% RSLogix 500 project LINCE050116_TOP.RSS, saved by version 11.00.00.00 %
PROJECT "LINCETOP"    % processor: MicroLogix 1400 %

PROGRAM FILES
  LAD 2 "MAIN"  12 rungs  % Main Program Routine %
  LAD 70 "OFFSETS"  43 rungs
  LAD 88 "TIMESWITCH"  2 rungs
  LAD 89 "SECONDS"  2 rungs
  LAD 90 "HSC"  9 rungs
  LAD 99 "HMI SET"  3 rungs
  LAD 100 "STI"  55 rungs
  LAD 102 "SPEED"  6 rungs
  LAD 104 "P ADJUST"  8 rungs
  LAD 110 "SHIFT"  11 rungs
  LAD 120 "XFER IN"  3 rungs
  LAD 121 "SIM PARTS"  7 rungs
  LAD 122 "PARTDETECT"  12 rungs
  LAD 123 "OPTICWIDTH"  7 rungs
  LAD 124 "PART GAP"  8 rungs
  LAD 125 "OPTIC CL"  4 rungs
  LAD 126 "ALIGNMENT"  6 rungs
  LAD 127 "OPTIC_LOAD"  3 rungs
  LAD 128 "FELL PART"  12 rungs
  LAD 130 "INS 5 TRIG"  14 rungs
  LAD 131 "INS 5 RSLT"  18 rungs
  LAD 140 "INS 6 TRIG"  9 rungs
  LAD 141 "INS 6 RSLT"  18 rungs
  LAD 150 "INS 7 TRIG"  9 rungs
  LAD 151 "INS 7 RSLT"  18 rungs
  LAD 170 "PASSBLOW"  12 rungs
  LAD 180 "RECERK"  10 rungs
  LAD 200 "PRODRATE"  1 rungs
  LAD 230 "HMI GET"  1 rungs

DATA FILES
  O0 OUTPUT  6 elements
  I1 INPUT  8 elements
  S2 STATUS  66 elements
  B3 BINARY  14 elements
  T4 TIMER  40 elements
  C5 COUNTER  1 elements
  R6 CONTROL  14 elements
  N7 INTEGER  200 elements
  F8 FLOAT  100 elements
  B9 TOP BS DAT  256 elements
  B10 TEMP  128 elements  % temp for program change %
  B11 TOP ER DAT  256 elements
  N12 TEMP  128 elements  % until sort out program io difference %
  L13  COUNTS  100 elements
  L23 NEW READ  100 elements
  L24 NEW WRITE  100 elements
  L42   52 elements
  B181 BLANK  128 elements  % used to wipe bs files %
  F182 TEST FLOAT  22 elements
  L183 TEST LONG  22 elements
  N184 TEST INTS  22 elements
  B185 TEST BITS  22 elements
  N186 HMI INTS  20 elements
  L187 HMI LONG  22 elements
  F188 HMI FLOATS  20 elements
  B189 HMI BITS  20 elements
  L190 COUNTS  128 elements
  B191 ERROR BITS  10 elements
  L192 SPD OFFSET  55 elements
  F193 SPD OFFSET  55 elements
  B194 GOOD BS  256 elements
  B195 NOERROR BS  256 elements
  B196 CTRL BITS  50 elements
  N197 CTRL INTS  50 elements
  B198 TRK BITS  50 elements
  L199 TRK LNG  50 elements
  N200 TRK INTS  50 elements
  L201 INS LNG  50 elements
  B202 INS BITS  50 elements
  N203 INS INTS  50 elements
  L204 CTRL LONG  60 elements
  F205 CTRL FLTS  50 elements

LADDER 2 "MAIN"    % Main Program Routine %
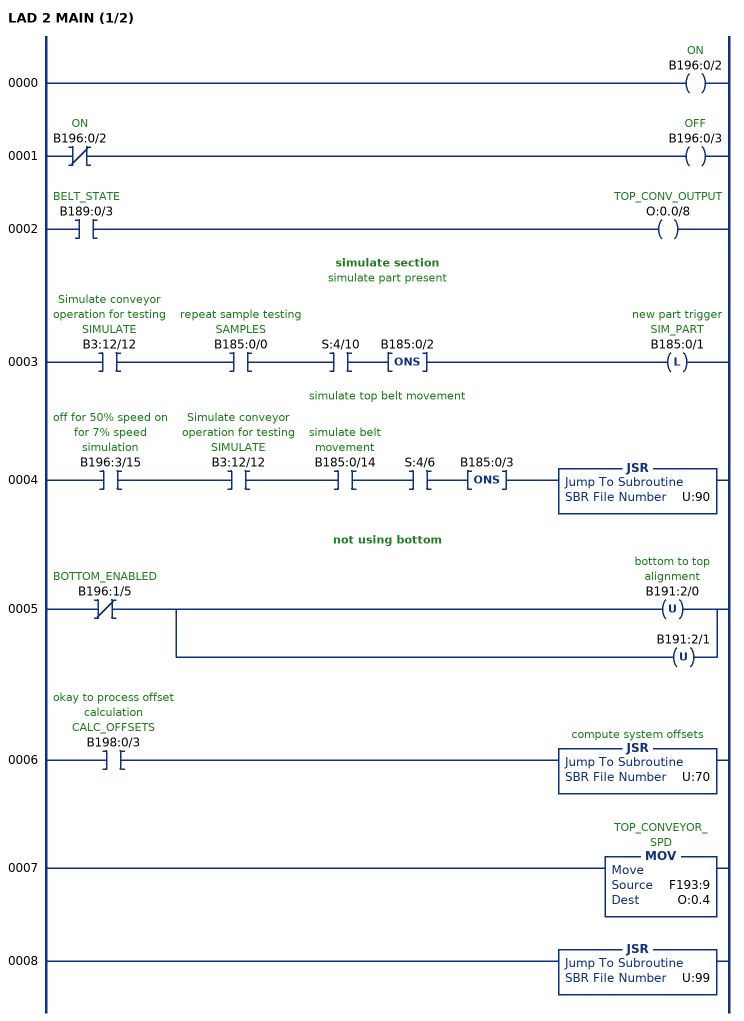
% Rung: 0 %
SOR OTE B196:0/2 EOR
%   B196:0/2  ON %
% Rung: 1 %
SOR XIO B196:0/2 OTE B196:0/3 EOR
%   B196:0/2  ON %
%   B196:0/3  OFF %
% Rung: 2 %
SOR XIC B189:0/3 OTE O:0.0/8 EOR
%   B189:0/3  BELT_STATE %
%   O:0.0/8  TOP_CONV_OUTPUT %
% Rung: 3 %
% TITLE: simulate section %
% simulate part present %
SOR XIC B3:12/12 XIC B185:0/0 XIC S:4/10 ONS B185:0/2 OTL B185:0/1 EOR
%   B3:12/12  SIMULATE  "Simulate conveyor operation for testing" %
%   B185:0/0  SAMPLES  "repeat sample testing" %
%   B185:0/1  SIM_PART  "new part trigger" %
% Rung: 4 %
% simulate top belt movement %
SOR XIC B196:3/15 XIC B3:12/12 XIC B185:0/14 XIC S:4/6 ONS B185:0/3 JSR U:90 EOR
%   B196:3/15  "off for 50% speed on for 7% speed simulation" %
%   B3:12/12  SIMULATE  "Simulate conveyor operation for testing" %
%   B185:0/14  "simulate belt movement" %
% Rung: 5 %
% TITLE: not using bottom %
SOR XIO B196:1/5 BST OTU B191:2/0 NXB OTU B191:2/1 BND EOR
%   B196:1/5  BOTTOM_ENABLED %
%   B191:2/0  "bottom to top alignment" %
% Rung: 6 %
SOR XIC B198:0/3 JSR U:70 EOR
%   B198:0/3  CALC_OFFSETS  "okay to process offset calculation" %
%   U:70  "compute system offsets" %
% Rung: 7 %
SOR MOV F193:9 O:0.4 EOR
%   F193:9  CTRLED_SCALED_VALUE %
%   O:0.4  TOP_CONVEYOR_SPD %
% Rung: 8 %
SOR JSR U:99 EOR

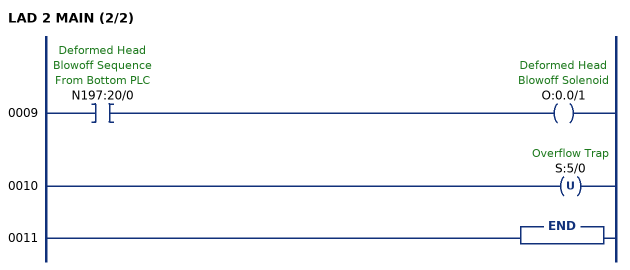
% Rung: 9 %
SOR XIC N197:20/0 OTE O:0.0/1 EOR
%   N197:20/0  "Deformed Head Blowoff Sequence From Bottom PLC" %
%   O:0.0/1  "Deformed Head Blowoff Solenoid" %
% Rung: 10 %
SOR OTU S:5/0 EOR
%   S:5/0  "Overflow Trap" %
% Rung: 11 %
SOR END EOR

LADDER 70 "OFFSETS"
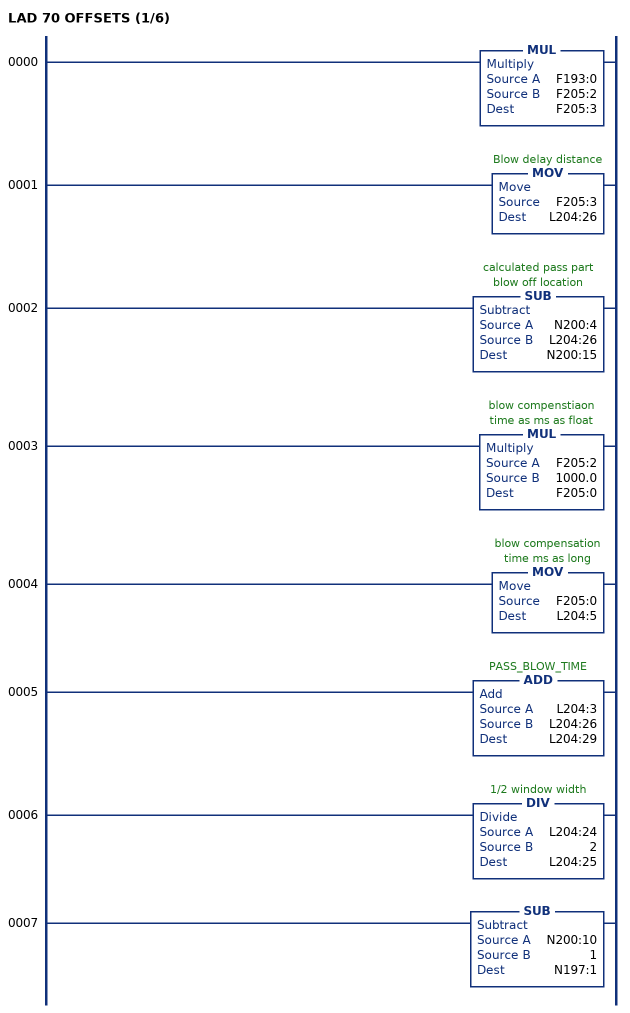
% Rung: 0 %
SOR MUL F193:0 F205:2 F205:3 EOR
%   F193:0  SPD  "speed calculation result (PPS)" %
%   F205:2  "blow compensation delay time from hmi" %
% Rung: 1 %
SOR MOV F205:3 L204:26 EOR
%   L204:26  "Blow delay distance" %
% Rung: 2 %
SOR SUB N200:4 L204:26 N200:15 EOR
%   N200:4  PASS_BLOW_LOC %
%   L204:26  "Blow delay distance" %
%   N200:15  "calculated pass part blow off location" %
% Rung: 3 %
SOR MUL F205:2 1000.0 F205:0 EOR
%   F205:2  "blow compensation delay time from hmi" %
%   F205:0  "blow compenstiaon time as ms as float" %
% Rung: 4 %
SOR MOV F205:0 L204:5 EOR
%   F205:0  "blow compenstiaon time as ms as float" %
%   L204:5  "blow compensation time ms as long" %
% Rung: 5 %
SOR ADD L204:3 L204:26 L204:29 EOR
%   L204:3  "blow on time" %
%   L204:26  "Blow delay distance" %
%   L204:29  PASS_BLOW_TIME %
% Rung: 6 %
SOR DIV L204:24 2 L204:25 EOR
%   L204:24  "window width" %
%   L204:25  "1/2 window width" %
% Rung: 7 %
SOR SUB N200:10 1 N197:1 EOR
%   N200:10  "Recirc Sensor Position" %

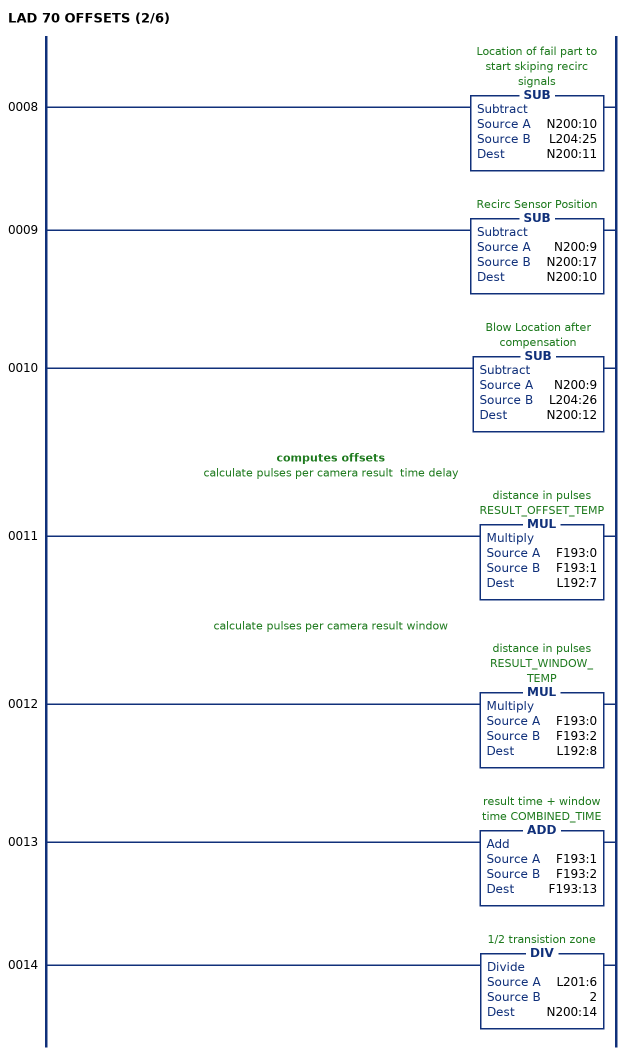
% Rung: 8 %
SOR SUB N200:10 L204:25 N200:11 EOR
%   N200:10  "Recirc Sensor Position" %
%   L204:25  "1/2 window width" %
%   N200:11  "Location of fail part to start skiping recirc signals" %
% Rung: 9 %
SOR SUB N200:9 N200:17 N200:10 EOR
%   N200:9  RECERK_BLOW_LOC %
%   N200:10  "Recirc Sensor Position" %
% Rung: 10 %
SOR SUB N200:9 L204:26 N200:12 EOR
%   N200:9  RECERK_BLOW_LOC %
%   L204:26  "Blow delay distance" %
%   N200:12  "Blow Location after compensation" %
% Rung: 11 %
% TITLE: computes offsets %
% calculate pulses per camera result  time delay %
SOR MUL F193:0 F193:1 L192:7 EOR
%   F193:0  SPD  "speed calculation result (PPS)" %
%   F193:1  RESULT_TIME_F  "Seconds" %
%   L192:7  RESULT_OFFSET_TEMP  "distance in pulses" %
% Rung: 12 %
% calculate pulses per camera result window %
SOR MUL F193:0 F193:2 L192:8 EOR
%   F193:0  SPD  "speed calculation result (PPS)" %
%   F193:2  WINDOW_TIME_F  "seconds" %
%   L192:8  RESULT_WINDOW_TEMP  "distance in pulses" %
% Rung: 13 %
SOR ADD F193:1 F193:2 F193:13 EOR
%   F193:1  RESULT_TIME_F  "Seconds" %
%   F193:2  WINDOW_TIME_F  "seconds" %
%   F193:13  COMBINED_TIME  "result time + window time" %
% Rung: 14 %
SOR DIV L201:6 2 N200:14 EOR
%   L201:6  OFFSET_MAX %
%   N200:14  "1/2 transistion zone" %

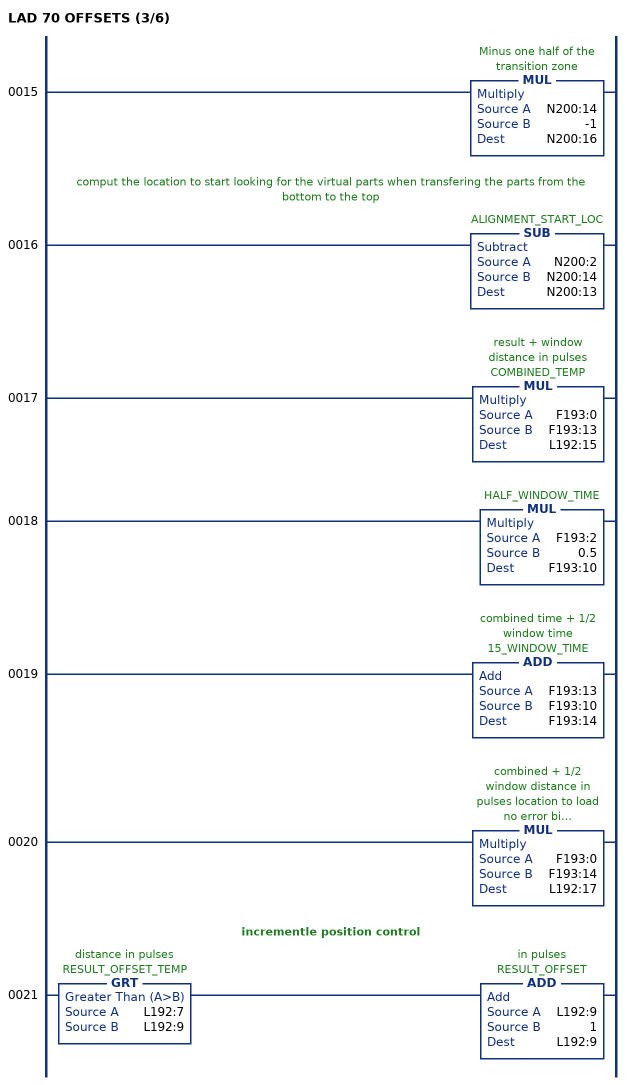
% Rung: 15 %
SOR MUL N200:14 -1 N200:16 EOR
%   N200:14  "1/2 transistion zone" %
%   N200:16  "Minus one half of the transition zone" %
% Rung: 16 %
% comput the location to start looking for the virtual parts when transfering the parts from the bottom to the top %
SOR SUB N200:2 N200:14 N200:13 EOR
%   N200:2  OPTIC_LOC %
%   N200:14  "1/2 transistion zone" %
%   N200:13  ALIGNMENT_START_LOC %
% Rung: 17 %
SOR MUL F193:0 F193:13 L192:15 EOR
%   F193:0  SPD  "speed calculation result (PPS)" %
%   F193:13  COMBINED_TIME  "result time + window time" %
%   L192:15  COMBINED_TEMP  "result + window distance in pulses" %
% Rung: 18 %
SOR MUL F193:2 0.5 F193:10 EOR
%   F193:2  WINDOW_TIME_F  "seconds" %
%   F193:10  HALF_WINDOW_TIME %
% Rung: 19 %
SOR ADD F193:13 F193:10 F193:14 EOR
%   F193:13  COMBINED_TIME  "result time + window time" %
%   F193:10  HALF_WINDOW_TIME %
%   F193:14  15_WINDOW_TIME  "combined time + 1/2 window time" %
% Rung: 20 %
SOR MUL F193:0 F193:14 L192:17 EOR
%   F193:0  SPD  "speed calculation result (PPS)" %
%   F193:14  15_WINDOW_TIME  "combined time + 1/2 window time" %
%   L192:17  15_WINDOW_TEMP  "combined + 1/2 window distance in pulses location to load no error bit" %
% Rung: 21 %
% TITLE: incrementle position control %
SOR GRT L192:7 L192:9 ADD L192:9 1 L192:9 EOR
%   L192:7  RESULT_OFFSET_TEMP  "distance in pulses" %
%   L192:9  RESULT_OFFSET  "in pulses" %

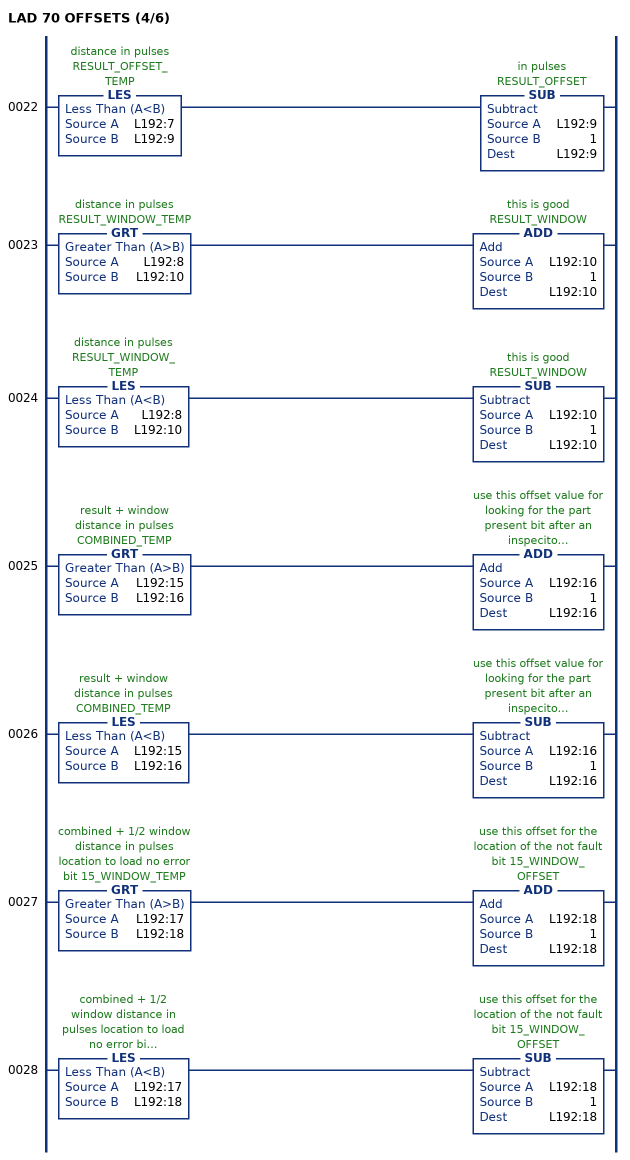
% Rung: 22 %
SOR LES L192:7 L192:9 SUB L192:9 1 L192:9 EOR
%   L192:7  RESULT_OFFSET_TEMP  "distance in pulses" %
%   L192:9  RESULT_OFFSET  "in pulses" %
% Rung: 23 %
SOR GRT L192:8 L192:10 ADD L192:10 1 L192:10 EOR
%   L192:8  RESULT_WINDOW_TEMP  "distance in pulses" %
%   L192:10  RESULT_WINDOW  "this is good" %
% Rung: 24 %
SOR LES L192:8 L192:10 SUB L192:10 1 L192:10 EOR
%   L192:8  RESULT_WINDOW_TEMP  "distance in pulses" %
%   L192:10  RESULT_WINDOW  "this is good" %
% Rung: 25 %
SOR GRT L192:15 L192:16 ADD L192:16 1 L192:16 EOR
%   L192:15  COMBINED_TEMP  "result + window distance in pulses" %
%   L192:16  COMBINED_OFFSET  "use this offset value for looking for the part present bit after an inspeciton" %
% Rung: 26 %
SOR LES L192:15 L192:16 SUB L192:16 1 L192:16 EOR
%   L192:15  COMBINED_TEMP  "result + window distance in pulses" %
%   L192:16  COMBINED_OFFSET  "use this offset value for looking for the part present bit after an inspeciton" %
% Rung: 27 %
SOR GRT L192:17 L192:18 ADD L192:18 1 L192:18 EOR
%   L192:17  15_WINDOW_TEMP  "combined + 1/2 window distance in pulses location to load no error bit" %
%   L192:18  15_WINDOW_OFFSET  "use this offset for the location of the not fault bit" %
% Rung: 28 %
SOR LES L192:17 L192:18 SUB L192:18 1 L192:18 EOR
%   L192:17  15_WINDOW_TEMP  "combined + 1/2 window distance in pulses location to load no error bit" %
%   L192:18  15_WINDOW_OFFSET  "use this offset for the location of the not fault bit" %

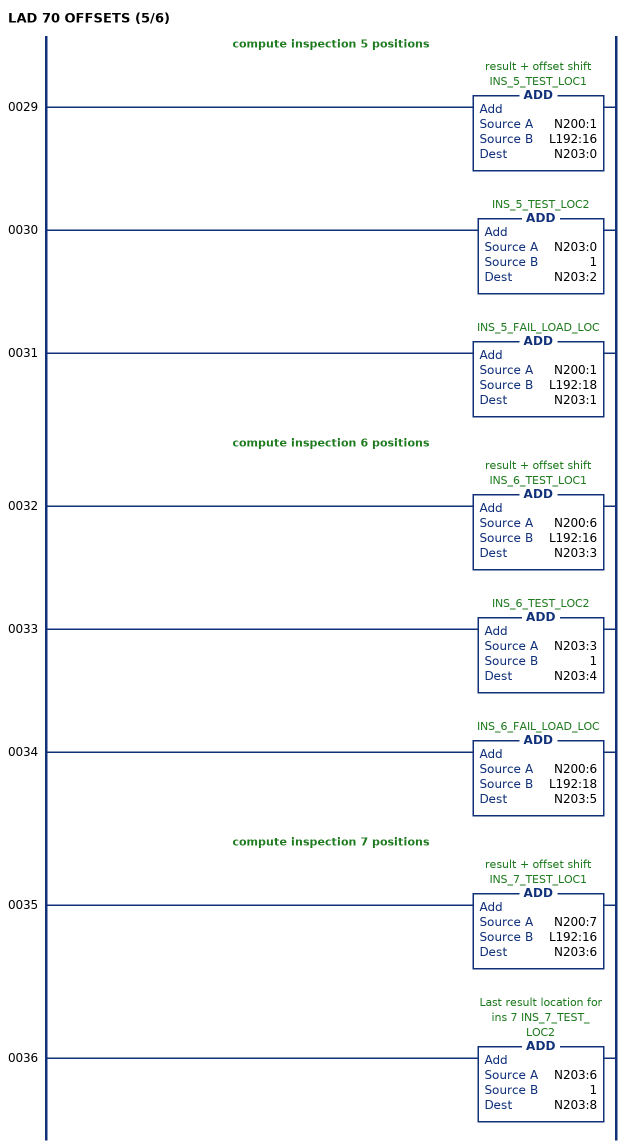
% Rung: 29 %
% TITLE: compute inspection 5 positions %
SOR ADD N200:1 L192:16 N203:0 EOR
%   N200:1  INS_5_TRIG_LOC %
%   L192:16  COMBINED_OFFSET  "use this offset value for looking for the part present bit after an inspeciton" %
%   N203:0  INS_5_TEST_LOC1  "result + offset shift" %
% Rung: 30 %
SOR ADD N203:0 1 N203:2 EOR
%   N203:0  INS_5_TEST_LOC1  "result + offset shift" %
%   N203:2  INS_5_TEST_LOC2 %
% Rung: 31 %
SOR ADD N200:1 L192:18 N203:1 EOR
%   N200:1  INS_5_TRIG_LOC %
%   L192:18  15_WINDOW_OFFSET  "use this offset for the location of the not fault bit" %
%   N203:1  INS_5_FAIL_LOAD_LOC %
% Rung: 32 %
% TITLE: compute inspection 6 positions %
SOR ADD N200:6 L192:16 N203:3 EOR
%   N200:6  INS_6_TRIG_LOC %
%   L192:16  COMBINED_OFFSET  "use this offset value for looking for the part present bit after an inspeciton" %
%   N203:3  INS_6_TEST_LOC1  "result + offset shift" %
% Rung: 33 %
SOR ADD N203:3 1 N203:4 EOR
%   N203:3  INS_6_TEST_LOC1  "result + offset shift" %
%   N203:4  INS_6_TEST_LOC2 %
% Rung: 34 %
SOR ADD N200:6 L192:18 N203:5 EOR
%   N200:6  INS_6_TRIG_LOC %
%   L192:18  15_WINDOW_OFFSET  "use this offset for the location of the not fault bit" %
%   N203:5  INS_6_FAIL_LOAD_LOC %
% Rung: 35 %
% TITLE: compute inspection 7 positions %
SOR ADD N200:7 L192:16 N203:6 EOR
%   N200:7  INS_7_TRIG_LOC %
%   L192:16  COMBINED_OFFSET  "use this offset value for looking for the part present bit after an inspeciton" %
%   N203:6  INS_7_TEST_LOC1  "result + offset shift" %
% Rung: 36 %
SOR ADD N203:6 1 N203:8 EOR
%   N203:6  INS_7_TEST_LOC1  "result + offset shift" %
%   N203:8  INS_7_TEST_LOC2  "Last result location for ins 7" %

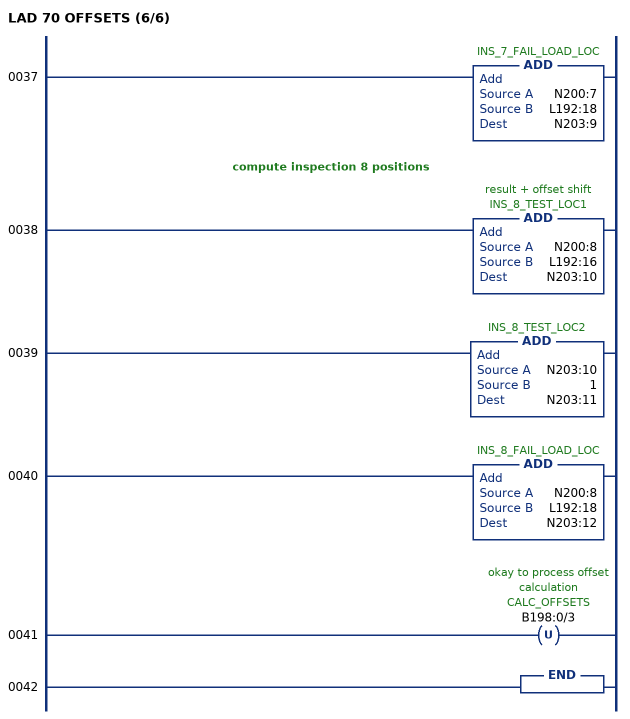
% Rung: 37 %
SOR ADD N200:7 L192:18 N203:9 EOR
%   N200:7  INS_7_TRIG_LOC %
%   L192:18  15_WINDOW_OFFSET  "use this offset for the location of the not fault bit" %
%   N203:9  INS_7_FAIL_LOAD_LOC %
% Rung: 38 %
% TITLE: compute inspection 8 positions %
SOR ADD N200:8 L192:16 N203:10 EOR
%   N200:8  INS_8_TRIG_LOC %
%   L192:16  COMBINED_OFFSET  "use this offset value for looking for the part present bit after an inspeciton" %
%   N203:10  INS_8_TEST_LOC1  "result + offset shift" %
% Rung: 39 %
SOR ADD N203:10 1 N203:11 EOR
%   N203:10  INS_8_TEST_LOC1  "result + offset shift" %
%   N203:11  INS_8_TEST_LOC2 %
% Rung: 40 %
SOR ADD N200:8 L192:18 N203:12 EOR
%   N200:8  INS_8_TRIG_LOC %
%   L192:18  15_WINDOW_OFFSET  "use this offset for the location of the not fault bit" %
%   N203:12  INS_8_FAIL_LOAD_LOC %
% Rung: 41 %
SOR OTU B198:0/3 EOR
%   B198:0/3  CALC_OFFSETS  "okay to process offset calculation" %
% Rung: 42 %
SOR END EOR

LADDER 88 "TIMESWITCH"
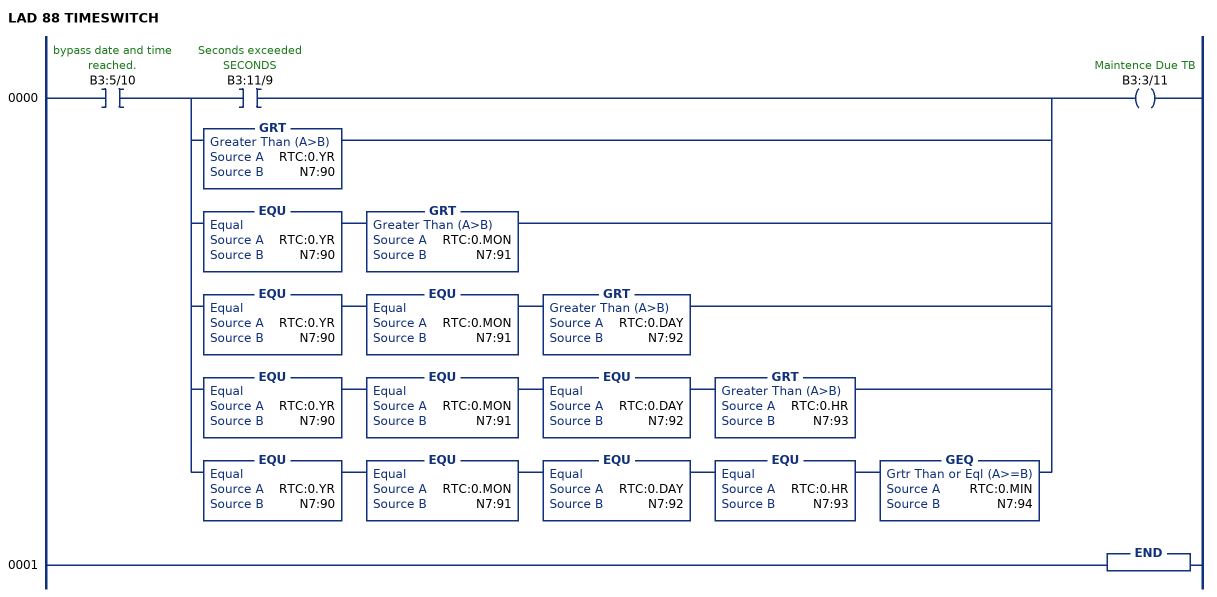
% Rung: 0 %
SOR XIC B3:5/10 BST XIC B3:11/9 NXB GRT RTC:0.YR N7:90 NXB EQU RTC:0.YR N7:90 GRT RTC:0.MON N7:91 NXB EQU RTC:0.YR N7:90 EQU RTC:0.MON N7:91 GRT RTC:0.DAY N7:92 NXB EQU RTC:0.YR N7:90 EQU RTC:0.MON N7:91 EQU RTC:0.DAY N7:92 GRT RTC:0.HR N7:93 NXB EQU RTC:0.YR N7:90 EQU RTC:0.MON N7:91 EQU RTC:0.DAY N7:92 EQU RTC:0.HR N7:93 GEQ RTC:0.MIN N7:94 BND OTE B3:3/11 EOR
%   B3:5/10  "bypass date and time reached." %
%   B3:11/9  SECONDS  "Seconds exceeded" %
%   N7:90  RTC %
%   B3:3/11  TB  "Maintence Due" %
% Rung: 1 %
SOR END EOR

LADDER 89 "SECONDS"
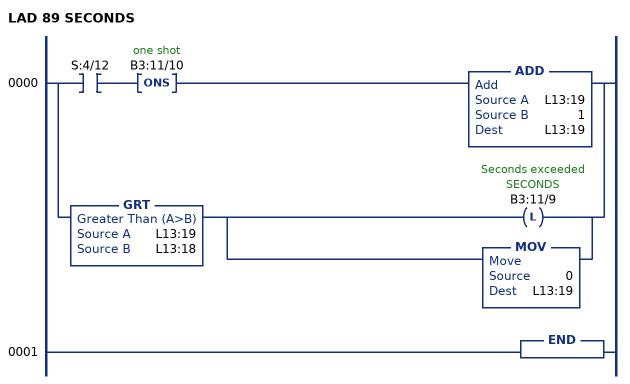
% Rung: 0 %
SOR BST XIC S:4/12 ONS B3:11/10 ADD L13:19 1 L13:19 NXB GRT L13:19 L13:18 BST OTL B3:11/9 NXB MOV 0 L13:19 BND BND EOR
%   B3:11/10  "one shot" %
%   L13:18  MAX %
%   B3:11/9  SECONDS  "Seconds exceeded" %
% Rung: 1 %
SOR END EOR

LADDER 90 "HSC"
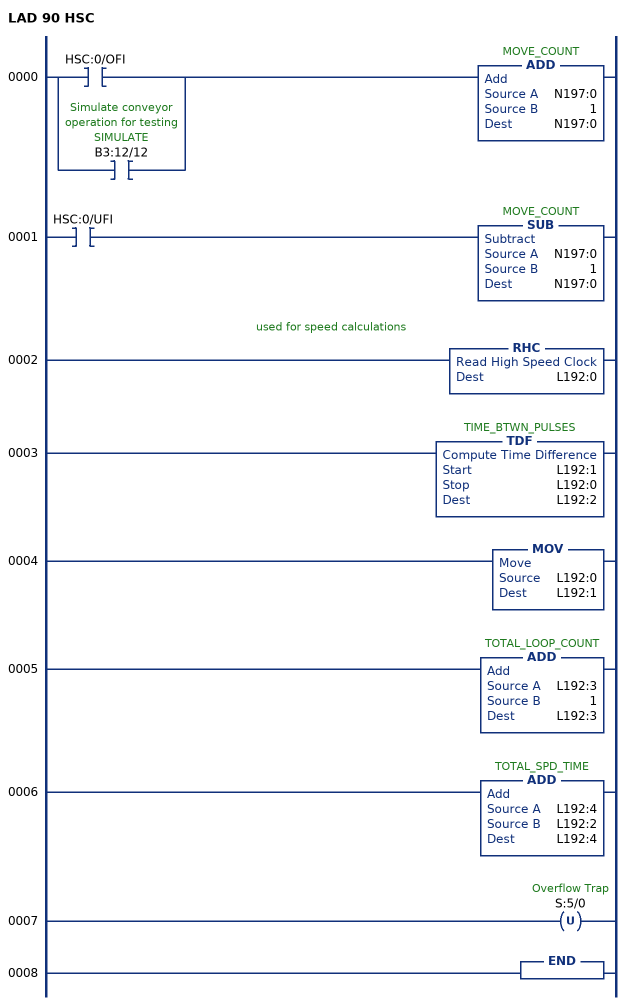
% Rung: 0 %
SOR BST XIC HSC:0/OFI NXB XIC B3:12/12 BND ADD N197:0 1 N197:0 EOR
%   B3:12/12  SIMULATE  "Simulate conveyor operation for testing" %
%   N197:0  MOVE_COUNT %
% Rung: 1 %
SOR XIC HSC:0/UFI SUB N197:0 1 N197:0 EOR
%   N197:0  MOVE_COUNT %
% Rung: 2 %
% used for speed calculations %
SOR RHC L192:0 EOR
% Rung: 3 %
SOR TDF L192:1 L192:0 L192:2 EOR
%   L192:2  TIME_BTWN_PULSES %
% Rung: 4 %
SOR MOV L192:0 L192:1 EOR
% Rung: 5 %
SOR ADD L192:3 1 L192:3 EOR
%   L192:3  TOTAL_LOOP_COUNT %
% Rung: 6 %
SOR ADD L192:4 L192:2 L192:4 EOR
%   L192:4  TOTAL_SPD_TIME %
%   L192:2  TIME_BTWN_PULSES %
% Rung: 7 %
SOR OTU S:5/0 EOR
%   S:5/0  "Overflow Trap" %
% Rung: 8 %
SOR END EOR

LADDER 99 "HMI SET"
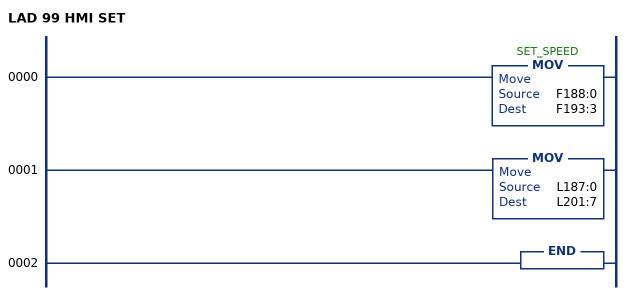
% Rung: 0 %
SOR MOV F188:0 F193:3 EOR
%   F188:0  HMI_SPEED  "hmi belt speed setting input" %
%   F193:3  SET_SPEED %
% Rung: 1 %
SOR MOV L187:0 L201:7 EOR
%   L187:0  ALIGN_OFFSET_MIN %
% Rung: 2 %
SOR END EOR

LADDER 100 "STI"
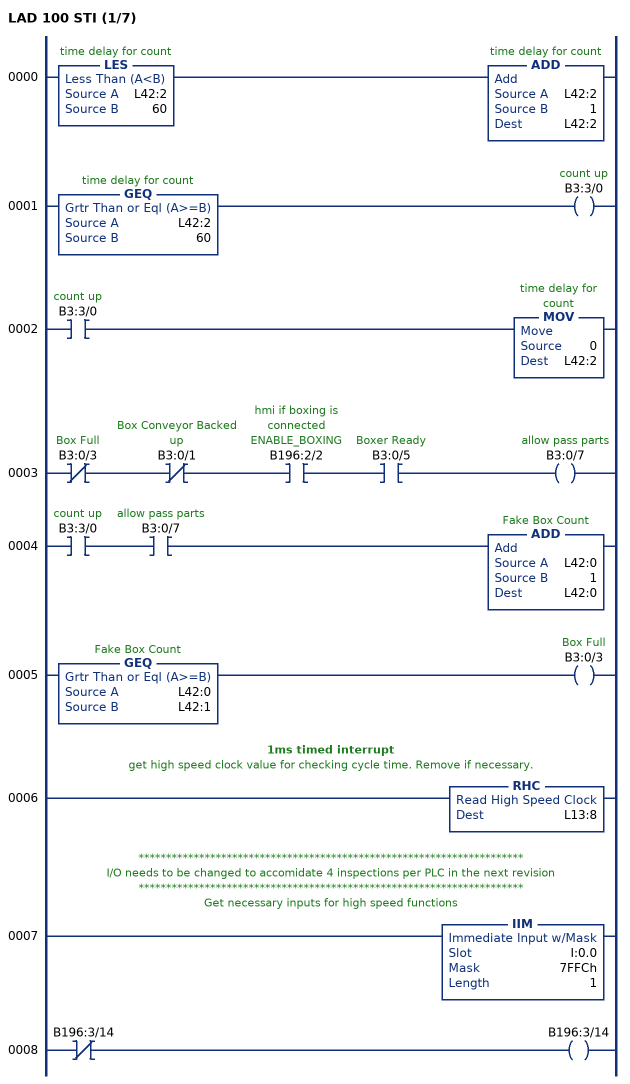
% Rung: 0 %
SOR LES L42:2 60 ADD L42:2 1 L42:2 EOR
%   L42:2  "time delay for count" %
% Rung: 1 %
SOR GEQ L42:2 60 OTE B3:3/0 EOR
%   L42:2  "time delay for count" %
%   B3:3/0  "count up" %
% Rung: 2 %
SOR XIC B3:3/0 MOV 0 L42:2 EOR
%   B3:3/0  "count up" %
%   L42:2  "time delay for count" %
% Rung: 3 %
SOR XIO B3:0/3 XIO B3:0/1 XIC B196:2/2 XIC B3:0/5 OTE B3:0/7 EOR
%   B3:0/3  "Box Full" %
%   B3:0/1  "Box Conveyor Backed up" %
%   B196:2/2  ENABLE_BOXING  "hmi if boxing is connected" %
%   B3:0/5  "Boxer Ready" %
%   B3:0/7  "allow pass parts" %
% Rung: 4 %
SOR XIC B3:3/0 XIC B3:0/7 ADD L42:0 1 L42:0 EOR
%   B3:3/0  "count up" %
%   B3:0/7  "allow pass parts" %
%   L42:0  "Fake Box Count" %
% Rung: 5 %
SOR GEQ L42:0 L42:1 OTE B3:0/3 EOR
%   L42:0  "Fake Box Count" %
%   L42:1  "Fake Box Limit" %
%   B3:0/3  "Box Full" %
% Rung: 6 %
% TITLE: 1ms timed interrupt %
% get high speed clock value for checking cycle time. Remove if necessary. %
SOR RHC L13:8 EOR
% Rung: 7 %
% **********************************************************************
% 
% I/O needs to be changed to accomidate 4 inspections per PLC in the next revision
% 
% **********************************************************************
% 
% Get necessary inputs for high speed functions %
SOR IIM I:0.0 7FFCh 1 EOR
% Rung: 8 %
SOR XIO B196:3/14 OTE B196:3/14 EOR

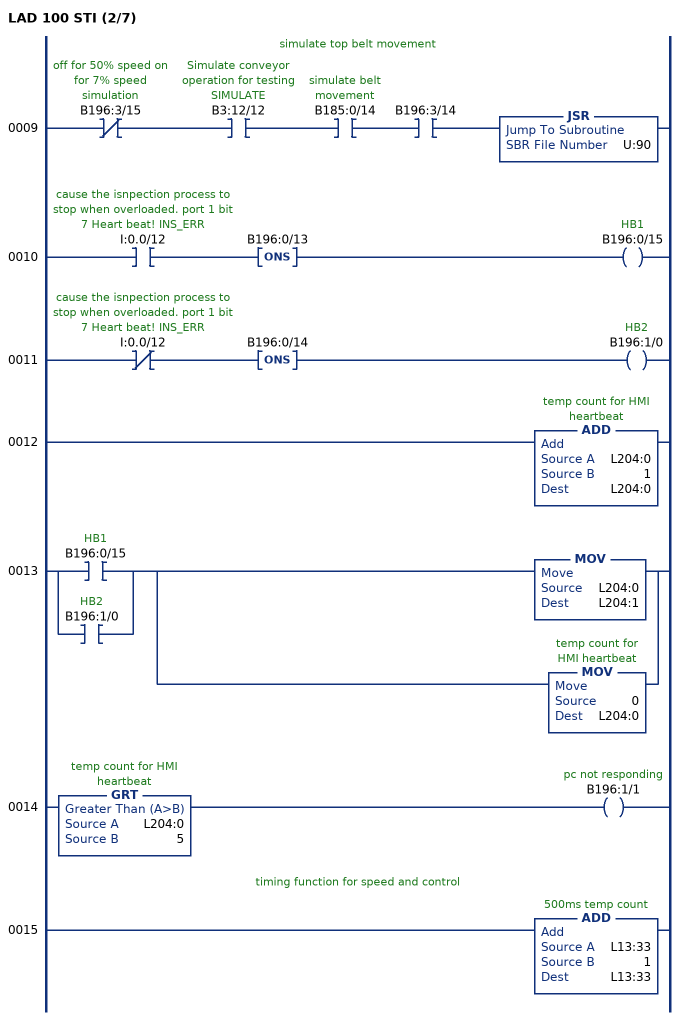
% Rung: 9 %
% simulate top belt movement %
SOR XIO B196:3/15 XIC B3:12/12 XIC B185:0/14 XIC B196:3/14 JSR U:90 EOR
%   B196:3/15  "off for 50% speed on for 7% speed simulation" %
%   B3:12/12  SIMULATE  "Simulate conveyor operation for testing" %
%   B185:0/14  "simulate belt movement" %
% Rung: 10 %
SOR XIC I:0.0/12 ONS B196:0/13 OTE B196:0/15 EOR
%   I:0.0/12  INS_ERR  "cause the isnpection process to stop when overloaded. port 1 bit 7 Heart beat!" %
%   B196:0/15  HB1 %
% Rung: 11 %
SOR XIO I:0.0/12 ONS B196:0/14 OTE B196:1/0 EOR
%   I:0.0/12  INS_ERR  "cause the isnpection process to stop when overloaded. port 1 bit 7 Heart beat!" %
%   B196:1/0  HB2 %
% Rung: 12 %
SOR ADD L204:0 1 L204:0 EOR
%   L204:0  "temp count for HMI heartbeat" %
% Rung: 13 %
SOR BST XIC B196:0/15 NXB XIC B196:1/0 BND BST MOV L204:0 L204:1 NXB MOV 0 L204:0 BND EOR
%   B196:0/15  HB1 %
%   B196:1/0  HB2 %
%   L204:0  "temp count for HMI heartbeat" %
% Rung: 14 %
SOR GRT L204:0 5 OTE B196:1/1 EOR
%   L204:0  "temp count for HMI heartbeat" %
%   B196:1/1  "pc not responding" %
% Rung: 15 %
% timing function for speed and control %
SOR ADD L13:33 1 L13:33 EOR
%   L13:33  "500ms temp count" %

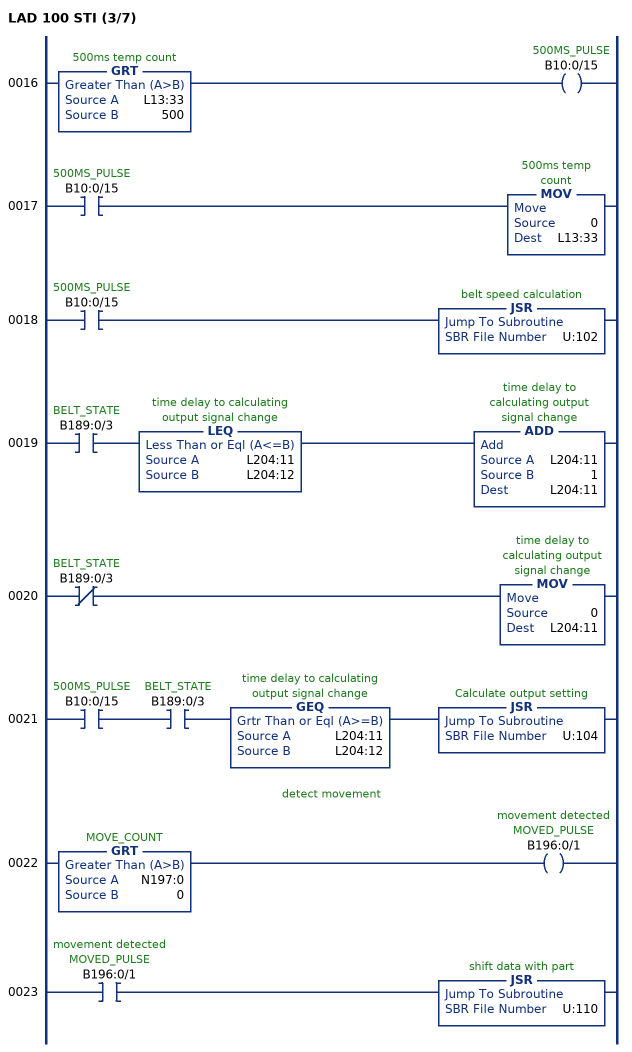
% Rung: 16 %
SOR GRT L13:33 500 OTE B10:0/15 EOR
%   L13:33  "500ms temp count" %
%   B10:0/15  500MS_PULSE %
% Rung: 17 %
SOR XIC B10:0/15 MOV 0 L13:33 EOR
%   B10:0/15  500MS_PULSE %
%   L13:33  "500ms temp count" %
% Rung: 18 %
SOR XIC B10:0/15 JSR U:102 EOR
%   B10:0/15  500MS_PULSE %
%   U:102  "belt speed calculation" %
% Rung: 19 %
SOR XIC B189:0/3 LEQ L204:11 L204:12 ADD L204:11 1 L204:11 EOR
%   B189:0/3  BELT_STATE %
%   L204:11  "time delay to calculating output signal change" %
% Rung: 20 %
SOR XIO B189:0/3 MOV 0 L204:11 EOR
%   B189:0/3  BELT_STATE %
%   L204:11  "time delay to calculating output signal change" %
% Rung: 21 %
SOR XIC B10:0/15 XIC B189:0/3 GEQ L204:11 L204:12 JSR U:104 EOR
%   B10:0/15  500MS_PULSE %
%   B189:0/3  BELT_STATE %
%   L204:11  "time delay to calculating output signal change" %
%   U:104  "Calculate output setting" %
% Rung: 22 %
% detect movement %
SOR GRT N197:0 0 OTE B196:0/1 EOR
%   N197:0  MOVE_COUNT %
%   B196:0/1  MOVED_PULSE  "movement detected" %
% Rung: 23 %
SOR XIC B196:0/1 JSR U:110 EOR
%   B196:0/1  MOVED_PULSE  "movement detected" %
%   U:110  "shift data with part" %

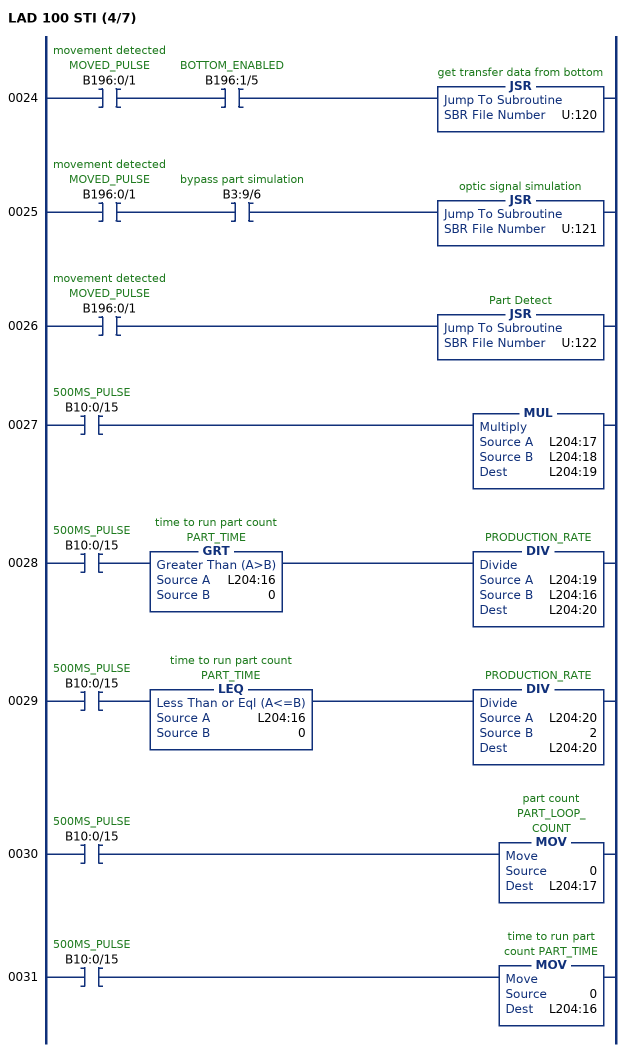
% Rung: 24 %
SOR XIC B196:0/1 XIC B196:1/5 JSR U:120 EOR
%   B196:0/1  MOVED_PULSE  "movement detected" %
%   B196:1/5  BOTTOM_ENABLED %
%   U:120  "get transfer data from bottom" %
% Rung: 25 %
SOR XIC B196:0/1 XIC B3:9/6 JSR U:121 EOR
%   B196:0/1  MOVED_PULSE  "movement detected" %
%   B3:9/6  "bypass part simulation" %
%   U:121  "optic signal simulation" %
% Rung: 26 %
SOR XIC B196:0/1 JSR U:122 EOR
%   B196:0/1  MOVED_PULSE  "movement detected" %
%   U:122  "Part Detect" %
% Rung: 27 %
SOR XIC B10:0/15 MUL L204:17 L204:18 L204:19 EOR
%   B10:0/15  500MS_PULSE %
%   L204:17  PART_LOOP_COUNT  "part count" %
% Rung: 28 %
SOR XIC B10:0/15 GRT L204:16 0 DIV L204:19 L204:16 L204:20 EOR
%   B10:0/15  500MS_PULSE %
%   L204:16  PART_TIME  "time to run part count" %
%   L204:20  PRODUCTION_RATE %
% Rung: 29 %
SOR XIC B10:0/15 LEQ L204:16 0 DIV L204:20 2 L204:20 EOR
%   B10:0/15  500MS_PULSE %
%   L204:16  PART_TIME  "time to run part count" %
%   L204:20  PRODUCTION_RATE %
% Rung: 30 %
SOR XIC B10:0/15 MOV 0 L204:17 EOR
%   B10:0/15  500MS_PULSE %
%   L204:17  PART_LOOP_COUNT  "part count" %
% Rung: 31 %
SOR XIC B10:0/15 MOV 0 L204:16 EOR
%   B10:0/15  500MS_PULSE %
%   L204:16  PART_TIME  "time to run part count" %

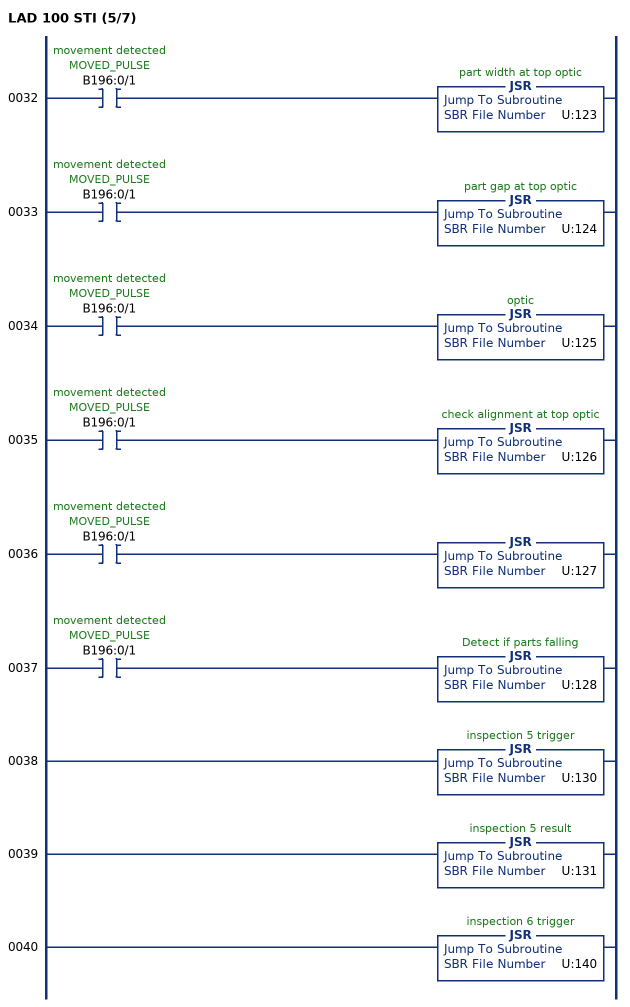
% Rung: 32 %
SOR XIC B196:0/1 JSR U:123 EOR
%   B196:0/1  MOVED_PULSE  "movement detected" %
%   U:123  "part width at top optic" %
% Rung: 33 %
SOR XIC B196:0/1 JSR U:124 EOR
%   B196:0/1  MOVED_PULSE  "movement detected" %
%   U:124  "part gap at top optic" %
% Rung: 34 %
SOR XIC B196:0/1 JSR U:125 EOR
%   B196:0/1  MOVED_PULSE  "movement detected" %
%   U:125  "optic" %
% Rung: 35 %
SOR XIC B196:0/1 JSR U:126 EOR
%   B196:0/1  MOVED_PULSE  "movement detected" %
%   U:126  "check alignment at top optic" %
% Rung: 36 %
SOR XIC B196:0/1 JSR U:127 EOR
%   B196:0/1  MOVED_PULSE  "movement detected" %
% Rung: 37 %
SOR XIC B196:0/1 JSR U:128 EOR
%   B196:0/1  MOVED_PULSE  "movement detected" %
%   U:128  "Detect if parts falling" %
% Rung: 38 %
SOR JSR U:130 EOR
%   U:130  "inspection 5 trigger" %
% Rung: 39 %
SOR JSR U:131 EOR
%   U:131  "inspection 5 result" %
% Rung: 40 %
SOR JSR U:140 EOR
%   U:140  "inspection 6 trigger" %

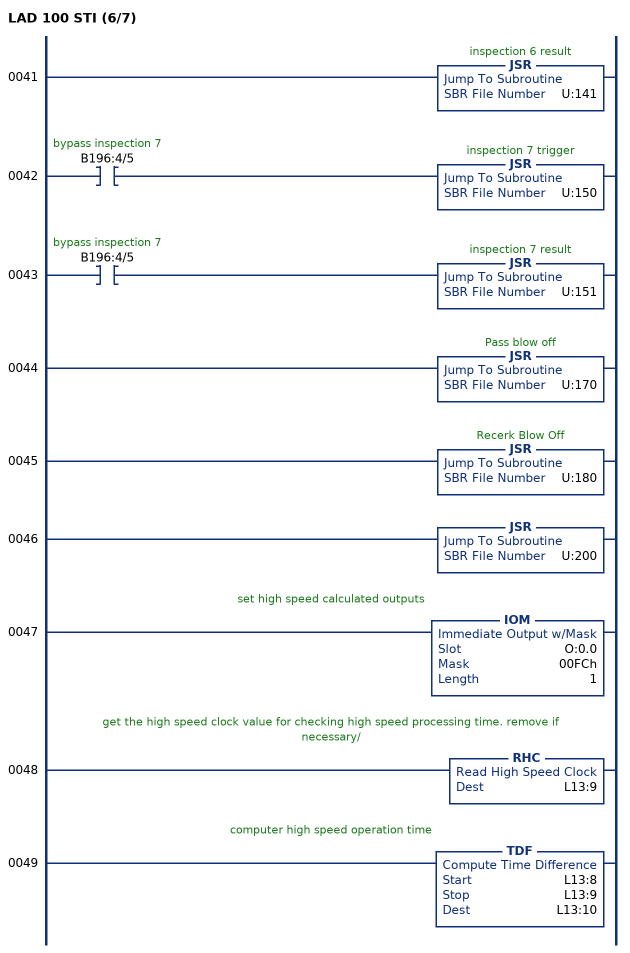
% Rung: 41 %
SOR JSR U:141 EOR
%   U:141  "inspection 6 result" %
% Rung: 42 %
SOR XIC B196:4/5 JSR U:150 EOR
%   B196:4/5  "bypass inspection 7" %
%   U:150  "inspection 7 trigger" %
% Rung: 43 %
SOR XIC B196:4/5 JSR U:151 EOR
%   B196:4/5  "bypass inspection 7" %
%   U:151  "inspection 7 result" %
% Rung: 44 %
SOR JSR U:170 EOR
%   U:170  "Pass blow off" %
% Rung: 45 %
SOR JSR U:180 EOR
%   U:180  "Recerk Blow Off" %
% Rung: 46 %
SOR JSR U:200 EOR
% Rung: 47 %
% set high speed calculated outputs %
SOR IOM O:0.0 00FCh 1 EOR
% Rung: 48 %
% get the high speed clock value for checking high speed processing time. remove if necessary/ %
SOR RHC L13:9 EOR
% Rung: 49 %
% computer high speed operation time %
SOR TDF L13:8 L13:9 L13:10 EOR

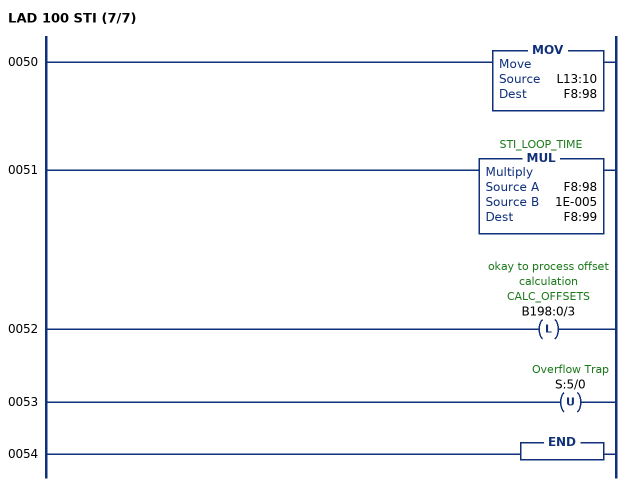
% Rung: 50 %
SOR MOV L13:10 F8:98 EOR
% Rung: 51 %
SOR MUL F8:98 1E-005 F8:99 EOR
%   F8:99  STI_LOOP_TIME %
% Rung: 52 %
SOR OTL B198:0/3 EOR
%   B198:0/3  CALC_OFFSETS  "okay to process offset calculation" %
% Rung: 53 %
SOR OTU S:5/0 EOR
%   S:5/0  "Overflow Trap" %
% Rung: 54 %
SOR END EOR

LADDER 102 "SPEED"
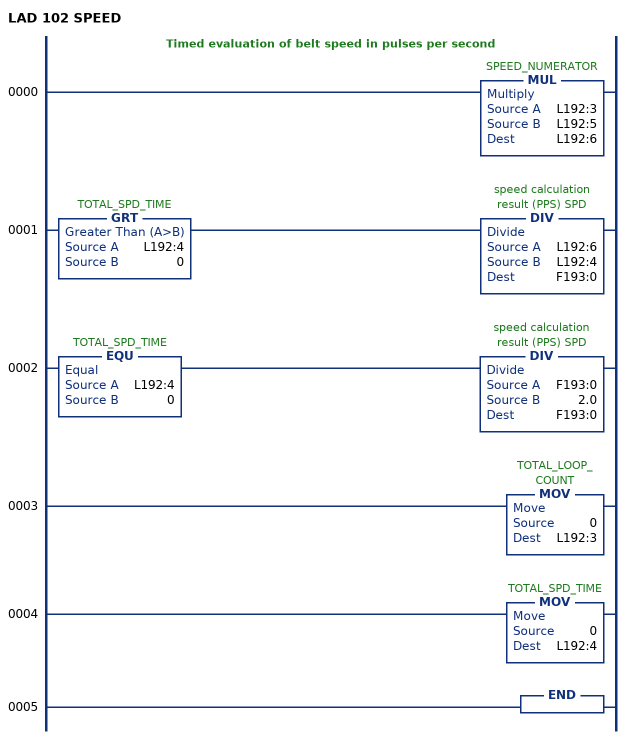
% Rung: 0 %
% TITLE: Timed evaluation of belt speed in pulses per second %
SOR MUL L192:3 L192:5 L192:6 EOR
%   L192:3  TOTAL_LOOP_COUNT %
%   L192:5  TKS_PER_SECOND %
%   L192:6  SPEED_NUMERATOR %
% Rung: 1 %
SOR GRT L192:4 0 DIV L192:6 L192:4 F193:0 EOR
%   L192:4  TOTAL_SPD_TIME %
%   L192:6  SPEED_NUMERATOR %
%   F193:0  SPD  "speed calculation result (PPS)" %
% Rung: 2 %
SOR EQU L192:4 0 DIV F193:0 2.0 F193:0 EOR
%   L192:4  TOTAL_SPD_TIME %
%   F193:0  SPD  "speed calculation result (PPS)" %
% Rung: 3 %
SOR MOV 0 L192:3 EOR
%   L192:3  TOTAL_LOOP_COUNT %
% Rung: 4 %
SOR MOV 0 L192:4 EOR
%   L192:4  TOTAL_SPD_TIME %
% Rung: 5 %
SOR END EOR

LADDER 104 "P ADJUST"
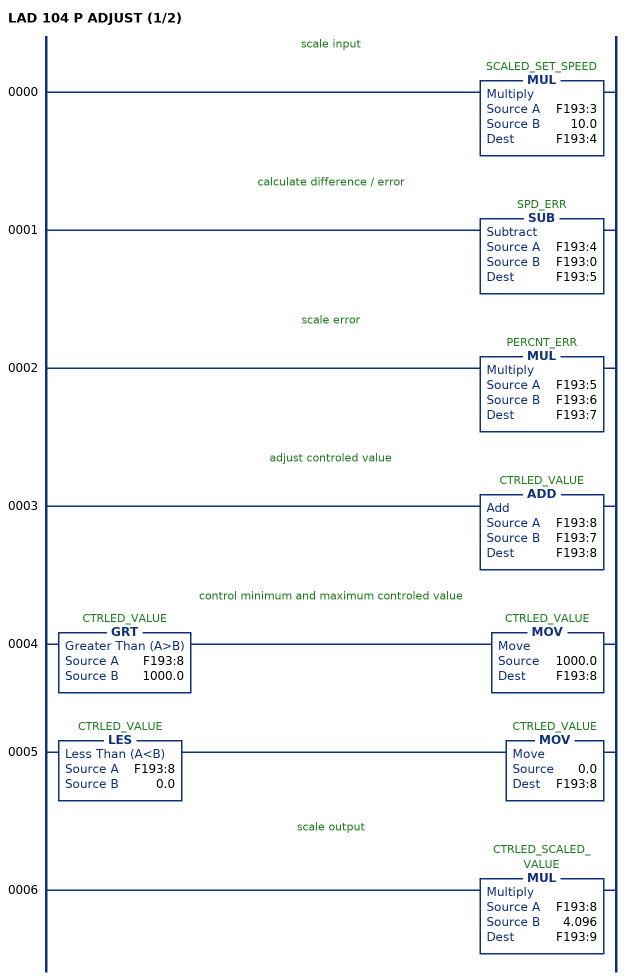
% Rung: 0 %
% scale input %
SOR MUL F193:3 10.0 F193:4 EOR
%   F193:3  SET_SPEED %
%   F193:4  SCALED_SET_SPEED %
% Rung: 1 %
% calculate difference / error %
SOR SUB F193:4 F193:0 F193:5 EOR
%   F193:4  SCALED_SET_SPEED %
%   F193:0  SPD  "speed calculation result (PPS)" %
%   F193:5  SPD_ERR %
% Rung: 2 %
% scale error %
SOR MUL F193:5 F193:6 F193:7 EOR
%   F193:5  SPD_ERR %
%   F193:6  FDBK_RATIO %
%   F193:7  PERCNT_ERR %
% Rung: 3 %
% adjust controled value %
SOR ADD F193:8 F193:7 F193:8 EOR
%   F193:8  CTRLED_VALUE %
%   F193:7  PERCNT_ERR %
% Rung: 4 %
% control minimum and maximum controled value %
SOR GRT F193:8 1000.0 MOV 1000.0 F193:8 EOR
%   F193:8  CTRLED_VALUE %
% Rung: 5 %
SOR LES F193:8 0.0 MOV 0.0 F193:8 EOR
%   F193:8  CTRLED_VALUE %
% Rung: 6 %
% scale output %
SOR MUL F193:8 4.096 F193:9 EOR
%   F193:8  CTRLED_VALUE %
%   F193:9  CTRLED_SCALED_VALUE %

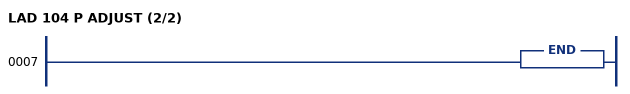
% Rung: 7 %
SOR END EOR

LADDER 110 "SHIFT"
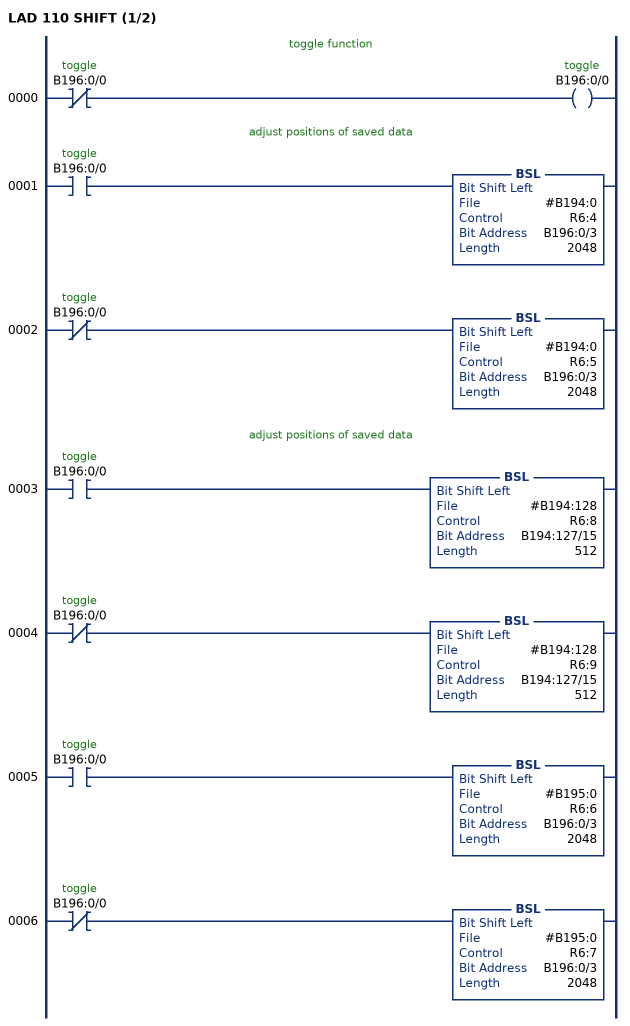
% Rung: 0 %
% toggle function %
SOR XIO B196:0/0 OTE B196:0/0 EOR
%   B196:0/0  "toggle" %
% Rung: 1 %
% adjust positions of saved data %
SOR XIC B196:0/0 BSL #B194:0 R6:4 B196:0/3 2048 EOR
%   B196:0/0  "toggle" %
%   B196:0/3  OFF %
% Rung: 2 %
SOR XIO B196:0/0 BSL #B194:0 R6:5 B196:0/3 2048 EOR
%   B196:0/0  "toggle" %
%   B196:0/3  OFF %
% Rung: 3 %
% adjust positions of saved data %
SOR XIC B196:0/0 BSL #B194:128 R6:8 B194:127/15 512 EOR
%   B196:0/0  "toggle" %
% Rung: 4 %
SOR XIO B196:0/0 BSL #B194:128 R6:9 B194:127/15 512 EOR
%   B196:0/0  "toggle" %
% Rung: 5 %
SOR XIC B196:0/0 BSL #B195:0 R6:6 B196:0/3 2048 EOR
%   B196:0/0  "toggle" %
%   B196:0/3  OFF %
% Rung: 6 %
SOR XIO B196:0/0 BSL #B195:0 R6:7 B196:0/3 2048 EOR
%   B196:0/0  "toggle" %
%   B196:0/3  OFF %

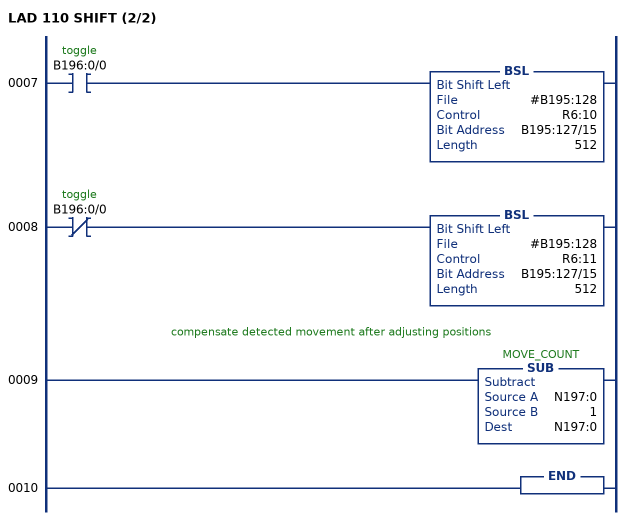
% Rung: 7 %
SOR XIC B196:0/0 BSL #B195:128 R6:10 B195:127/15 512 EOR
%   B196:0/0  "toggle" %
% Rung: 8 %
SOR XIO B196:0/0 BSL #B195:128 R6:11 B195:127/15 512 EOR
%   B196:0/0  "toggle" %
% Rung: 9 %
% compensate detected movement after adjusting positions %
SOR SUB N197:0 1 N197:0 EOR
%   N197:0  MOVE_COUNT %
% Rung: 10 %
SOR END EOR

LADDER 120 "XFER IN"
